// Mitsubishi GX Works2 project: counter+sequence_1   PLC: Q03UDV

PROGRAM MAIN
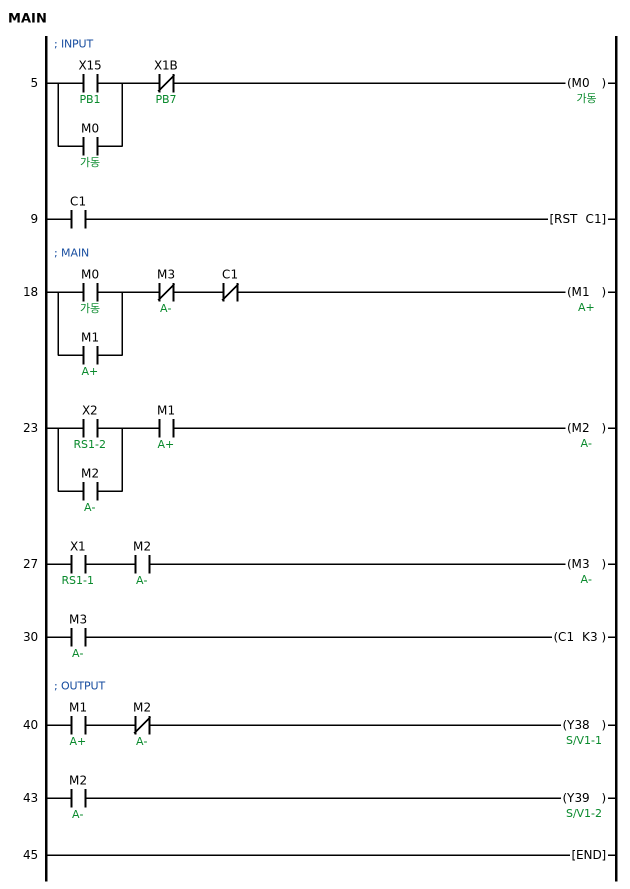
; INPUT
5     LD      X15  ; PB1
      OR      M0  ; 가동
      ANI     X1B  ; PB7
      OUT     M0  ; 가동
9     LD      C1
      RST     C1
; MAIN
18    LD      M0  ; 가동
      OR      M1  ; A+
      ANI     M3  ; A-
      ANI     C1
      OUT     M1  ; A+
23    LD      X2  ; RS1-2
      OR      M2  ; A-
      AND     M1  ; A+
      OUT     M2  ; A-
27    LD      X1  ; RS1-1
      AND     M2  ; A-
      OUT     M3  ; A-
30    LD      M3  ; A-
      OUT     C1 K3
; OUTPUT
40    LD      M1  ; A+
      ANI     M2  ; A-
      OUT     Y38  ; S/V1-1
43    LD      M2  ; A-
      OUT     Y39  ; S/V1-2
45    END
END_PROGRAM

// device comments not shown above
X3  ; RS2-1
X4  ; RS2-2
X16  ; PB2
X17  ; PB3
X18  ; PB4
M4  ; B-
M11  ; A+
M12  ; B+
M13  ; A-
M14  ; B-
M21  ; A+B+
M22  ; A-B-
M31  ; B+
M32  ; B-A+
M33  ; A-
Y3A  ; S/V2
